// TIA Portal V19 export
FUNCTION "FC_PAR_COPY" : Void   // FC55, STL
{ S7_Optimized_Access := 'FALSE' }
AUTHOR : MS
// Kopieren Rezeptparameter
// stored: AutoNumber false
   VAR_INPUT
      Pos_Nr : USInt;
      WT_DB_Nr : Word;
   END_VAR
   VAR_TEMP
      WT_DB : Word;
      Par_Nr : Int;
      Schrittweite : Int;
      Par_ID : USInt;
      Cmd : USInt;
   END_VAR
BEGIN

NETWORK
TITLE = Polwender verwenden
//Positionsadresse laden
      L     #Pos_Nr;
      L     0;
      ==I;
      BEC;

//WT DB laden
      L     #WT_DB_Nr;
      T     #WT_DB;
//Pointer auf Befehl 1 setzen
      OPN   DB [#WT_DB];
      L     %DBW0;  //max. Anzahl
      L     %DBW48;  //Befehls-Nr
      <=I;
      BEC;
      L     %DBW48;  //Befehls-Nr
      L     %DBW4;  //Länge
      *I;
      L     %DBW2;  //Offset
      +I;
      SLD   3;
      LAR1;
      L     DBB [AR1, P#0.0];  //akt_Cmd
      T     #Cmd;
      L     DBW [AR1, P#6.0];  //Param-Pntr
      T     %DBW46;  //Pointer aktuell

//------------------------
//Parameter Kopieren
//------------------------
      L     0;
      T     #Par_Nr;
RET:  L     #Pos_Nr;
      L     1;
      -I;
      L     "DB_PAR_ID".Leng;
      *I;
      L     "DB_PAR_ID".Offset;
      +I;
      L     #Par_Nr;
      +I;
      SLD   3;
      LAR1;
      OPN   "DB_PAR_ID";
      L     DBB [AR1, P#0.0];
      T     #Par_ID;
//PARAMETERADRESSE LADEN
      OPN   DB [#WT_DB];
      L     %DBW46;  //Pointer aktuell
      SLD   3;
      LAR2;

      OPN   "DB_POS";
      L     #Par_ID;
      JL    list;
      JU    ende;
      JU    ID1;  //1 Expozeit
      JU    ID2;  //2 Variante
list: JU    ende;
//------------------------------
//Sollexpo
//------------------------------
ID1:  L     4;
      T     #Schrittweite;

      L     1.0;
      L     "DB_POS".POS[0].KF_Expo;
      ==R;
      OPN   DB [#WT_DB];
      L     DBD [AR2, P#0.0];
      JC    ExOk;
      DTR;
      *R;
      RND;
ExOk: T     "DB_POS".POS[0].Soll_Expozeit;
      JU    NEXT;
//------------------------------
//Variante
//------------------------------
ID2:  L     1;
      T     #Schrittweite;
      JU    NEXT;

//-----------------------------
//nächsten Parameter laden
//-----------------------------
NEXT: OPN   DB [#WT_DB];
      L     %DBW46;
      L     #Schrittweite;
      +I;
      T     %DBW46;

      L     #Par_Nr;
      L     1;
      +I;
      T     #Par_Nr;
      L     "DB_PAR_ID".Leng;
      <I;
      JC    RET;
ende: BE;

END_FUNCTION
